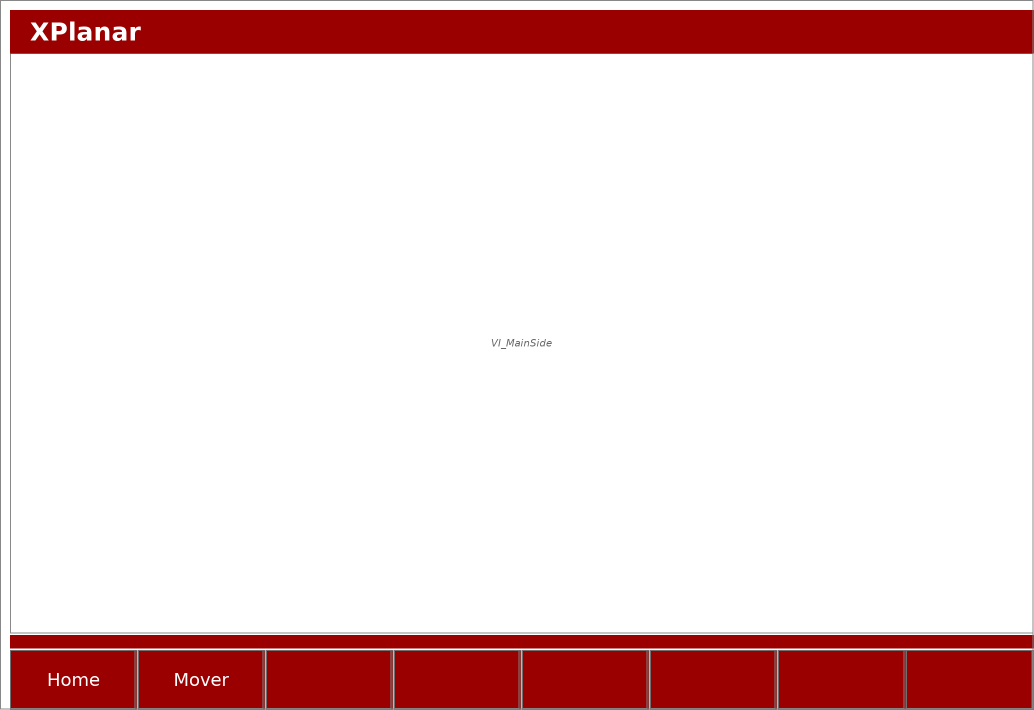
VISUALIZATION Visualization  // 1034x710
    Frame (10,53 1023x580)
        shows VI_MainSide()
        shows Tc3_XPlanarStandard.VI_MoverLogOverview()
        shows VI_EtherCatDiag()
        shows VI_MoverDiag()
        shows VI_MoverTuning()
        shows VI_MoverDiag()
        shows VI_Station()
        p1165984742: GVL_XtsVisu.pGroupRef[1]^.NcToPlc.Common.GroupStatus
        p547225198: GVL_XtsVisu.pGroupRef[1]
    Rectangle (10,10 1024x43), "XPlanar"
    Rectangle (10,635 1024x13)
    Button (10,650 127x60), "Home"
        OnMouseDown: FrameSelectionChange Selection=SelectedFrame=87eec691-4479-469a-bdd2-91ec7a1bb6bd, GlobSel=AssignType=Directly, SelType=Locally
    Button (138,650 127x60), "Mover"
        OnMouseUp: FrameSelectionChange Selection=SelectedFrame=87eec691-4479-469a-bdd2-91ec7a1bb6bd, Selection=1, GlobSel=AssignType=Directly, SelType=Locally
    Button (266,650 127x60)
    Button (394,650 127x60)
    Button (522,650 127x60)
    Button (650,650 127x60)
    Button (906,650 128x60)
    Button (778,650 128x60)
END_VISUALIZATION

(* stored: Version 1.1.0.1, ProductVersion 3.1.4024.9
   Visu Visualization: Id {9d7dad9d-1f08-40b5-aea6-4ac2b0d49e76} *)
